Fanuc KAREL source: KT00401.KL

PROGRAM KT00401
%NOLOCKGROUP
VAR
  I1: INTEGER
  I2: INTEGER
  OUT: BOOLEAN
BEGIN
  I1 = 2
  I2 = 3
  I1 = 2
  I2 = 3
  OUT = I1 > I2
END KT00401
